FUNCTION printChangeAxisEnable : BOOL
VAR_INPUT
	cmd: ChangeAxisEnable;
END_VAR
VAR
END_VAR

MSG.changeAxisEnable.ipArguments.Clear().AddDInt(cmd.axisIndex).AddBool(cmd.enabled);
MSG.changeAxisEnable.Send(0);

END_FUNCTION

(* stored: Version 1.1.0.1, ProductVersion 3.1.4022.12
   POU printChangeAxisEnable: Id {ef7a5dec-0803-41a2-bddf-34842043f831}, SpecialFunc None *)
